{attribute 'GeneratedUsingTerminal: ELM2742-0000-0016'}
{attribute addProperty BoxType "ELM2742-0000-0016"}
{attribute addProperty Id "EtcSlaveTerminalBaseDO_Inputs_DeviceAT %I*DO_Inputs_Device_4A9049C53DO_Group_1_OutputsAT %Q*DO_Group_1_Outputs_07009A9C4DO_Group_2_OutputsAT %Q*DO_Group_2_Outputs_3033EF654WcStateAT %I*WcState_9091E0EB2InfoDataAT %I*InfoData_BEF6B88E18"}
{attribute addProperty CRC "636260240"}
{attribute addProperty Size "31"}
TYPE ELM2742_25EC8F90 EXTENDS EtcSlaveTerminalBase :
STRUCT
	{attribute addProperty Name "DO_Inputs_Device"}
	DO_Inputs_Device : DO_Inputs_Device_4A9049C5;
	{attribute addProperty Name "DO_Group_1_Outputs"}
	DO_Group_1_Outputs : DO_Group_1_Outputs_07009A9C;
	{attribute addProperty Name "DO_Group_2_Outputs"}
	DO_Group_2_Outputs : DO_Group_2_Outputs_3033EF65;
	{attribute addProperty Name "WcState"}
	WcState : WcState_9091E0EB;
	{attribute addProperty Name "InfoData"}
	InfoData : InfoData_BEF6B88E;
END_STRUCT
END_TYPE

(* stored: Version 1.2.0.0, ProductVersion 3.1.4024.9
   DUT ELM2742_25EC8F90: Id {83fce538-c498-4f5e-9335-3bf2271654c9} *)
